// TIA Portal V20 export
// export: Created 2026-07-16T12:58:44.106145Z, ExportSetting WithDefaults, DisplayName Totally Integrated Automation Portal, DisplayVersion V20 Update 5, DisplayName TIA Portal Openness, DisplayVersion V20 Update 4, DisplayName TIA Portal Version Control Interface, DisplayVersion V20 Update 5, DisplayName SINAMICS Startdrive Advanced, DisplayVersion V20, DisplayName SINAMICS DCC, DisplayVersion V20, DisplayName SINAMICS Startdrive G130, G150, S120, S150, SINAMICS MV, G220, S200, S210, DisplayVersion V20, DisplayName SINAMICS Startdrive G110M, G120, G120C, G120D, G120P, G115D, DisplayVersion V20, DisplayName STEP 7 Professional, DisplayVersion V20 Update 5, DisplayName STEP 7 Safety, DisplayVersion V20 Update 2, DisplayName WinCC Basic/Comfort/Advanced, DisplayVersion V20 Update 5, DisplayName WinCC Unified, DisplayVersion V20 Update 5
DATA_BLOCK "DB_Input"   // DB1
{ S7_Optimized_Access := 'TRUE' }
VERSION : 0.1
// stored: AutoNumber true, DBAccessibleFromOPCUA true, IsOnlyStoredInLoadMemory false, IsRetainMemResEnabled false, IsWriteProtectedInAS false, MemoryReserve 100
   VAR
      Test : Array[0..22] of Bool;
      SpareDI : Array[1..7] of Bool;
      Control_Healthy : Bool;
      Cycle_Start : Bool;
      Cycle_Stop : Bool;
      Shredder_Run_Fwd_FB : Bool;
      Shredder_Run_Rev_FB : Bool;
      Motor_Fault : Bool;
      Hopper_Level_High : Bool;
      Infeed_Conv_Running : Bool;
      Discharge_Conv_Running : Bool;
      Pusher_PowerPack_Running : Bool;
      Pusher_Home_Limit : Bool;
      Pusher_Full_Travel_Limit : Bool;
      Pusher_High_Pressure : Bool;
      Downstream_Running : Bool;
      Pusher_Local_Remote : Bool;
   END_VAR
BEGIN
END_DATA_BLOCK
